Staubli VAL3: chkScaraFrame.pgx

program chkScaraFrame(frame x_frame (dimensions=1), num& x_nError[] (dimensions=1))
  local num l_nTeta
  local num l_nValueZ
  local point l_pOM
  local point l_pOrigin
begin
  // This program checks if the conveyor's frame is aligned to the robot
  // WORLD reference frame.
  // With a scara robot, the locations used to teach the conveyor's frame must have the
  // same altitude (Z coordinate) to build a frame aligned to the WORLD.
  // If not, the locations may not be reachable by the scara robot.
  //
  // Created 17-02-07                                   C.CURRIVAND
  //----------------------------------------------------------------
  //
  // Initialize local variables
  l_nValueZ=1000
  l_pOrigin=l_pOM=here(tPointer,world)
  //
  l_pOrigin.trsf={0,0,0,0,0,0}
  l_pOM=compose(l_pOrigin,x_frame,{0,0,l_nValueZ,0,0,0})
  //
  // Compute teta
  l_nTeta=atan(sqrt((l_pOM.trsf.x*l_pOM.trsf.x)+(l_pOM.trsf.y*l_pOM.trsf.y))/l_nValueZ)
  x_nError=sel(abs(l_nTeta)>1,1,0)
end
